{attribute 'no_explicit_call' := 'NormallyOpenSensor is a CLASS and must be accessed using methods or properties'}
FUNCTION_BLOCK NormallyOpenSensor
VAR
	input				AT %I*: BOOL;
END_VAR

PROPERTY IsActive : bool
GET
IsActive				:= not input;
END_GET
END_PROPERTY

PROPERTY IsNotActive : bool
GET
IsActive				:= input;
END_GET
END_PROPERTY

END_FUNCTION_BLOCK

(* stored: Version 1.1.0.1, ProductVersion 3.1.4024.11
   POU NormallyOpenSensor: Id {009a0b10-1ab5-4582-9cc8-968afc7fb534}, SpecialFunc None
   Property IsActive: Id {2a37620c-d5da-4012-826b-3868d05113fb}
   Get Get: Id {19a34990-c411-4e40-b2de-6c755d2e08c6}
   Property IsNotActive: Id {17dd950a-2c3b-464c-b165-865ca60ae828}
   Get Get: Id {1b02d1f0-0cdf-48d2-87c3-7a7214932ddb} *)
